(* CoDeSys 2.3 export: ALARMS.EXP *)

(* POU Alarm/ALARMS, ST *)
FUNCTION_BLOCK ALARMS
VAR_INPUT
	inReset: BOOL; (* Сброс зарегистрированых ошибок *)
END_VAR
VAR_OUTPUT
	outLastAlarm: INT; (* Номер последней ошибки *)
	outIsAlarm: BOOL; (* Есть ошибка для индикации *)
	outIsZoomer: BOOL; (* Есть ошибка для зумера *)
	outBlinker: BOOL; (* Мигает номер ошибки *)
	outAlarmCode :DWORD := 0;
END_VAR
VAR
	inResetM: BOOL; (* Память для сброса для определения фронта *)
	bCount: INT := 1; (* Счетчик для цикла*)

END_VAR
	(* Если есть сигнал сброса, сбрасываем общую регистрацию аварии, а так же номер последней аварии *)

	IF inReset AND NOT inResetM THEN
		ERR_RESET_ALL(inReset);
		outLastAlarm := 0;
	END_IF;

	inResetM := inReset;

	outIsAlarm  := outIsZoomer :=FALSE;

	(* Проверяем в цикле входящие ошибки *)

	FOR bCount := 1 TO _ERR_Nums DO

		(* Если есть авария, то назначаем состояние ощей аварии *)

		IF glbErrors[bCount].State OR glbErrors[bCount].LatchState THEN
			outIsAlarm := TRUE;
			outLastAlarm := bCount;
		END_IF;

		(* Включить зуммер если авария зарегистрирована и зуммер разрешен *)

		IF glbErrors[bCount].LatchState AND glbErrors[bCount].Zoomer THEN
			outIsZoomer  := TRUE;
		END_IF;

		IF glbErrors[bCount].State AND glbErrors[bCount].Zoomer THEN
			outIsZoomer  := TRUE;
		END_IF;

	END_FOR;

	outAlarmCode := ERR_CODE(
					glbErrors[1].State,
					glbErrors[2].State,
					glbErrors[3].State,
					glbErrors[4].State,
					glbErrors[5].State,
					glbErrors[6].State,
					glbErrors[7].State,
					glbErrors[8].State,
					glbErrors[9].State,
					glbErrors[10].State,
					glbErrors[11].State,
					glbErrors[12].State,
					glbErrors[13].State);
END_FUNCTION_BLOCK
